//Structure for specific subsystems related to an instrument
TYPE ST_SubSystemIn :
STRUCT
END_STRUCT
END_TYPE

(* stored: Version 1.1.0.1
   DUT ST_SubSystemIn: Id {aeb09d6b-ddca-03d8-0388-f1a06cf7485b} *)
